FUNCTION_BLOCK FB_Methods
VAR 
	
END_VAR

METHOD MethodDefaultValue
VAR_INPUT
	nValue1		: INT;
	nValue2		: INT := 5;
END_VAR
END_METHOD

END_FUNCTION_BLOCK

(* stored: Version 1.1.0.1, ProductVersion 3.1.4026.6
   POU FB_Methods: Id {6396cacb-4ab4-48c8-aa86-d49e12b23891}, SpecialFunc None
   Method MethodDefaultValue: Id {f032475f-3b96-49e8-b49b-354e07ef8f84} *)
